FUNCTION_BLOCK FB_DO (* Service Interface Function Block Type *)
  (* Standard: 61499-2 *)
  (* Version 0.0, 2014-5-4, wildai, nxtControl GmbH, template *)
  (* Compiler Cpp nxtControl builtin 1.0 *)
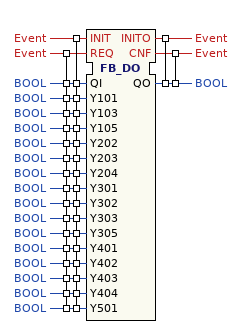
  EVENT_INPUT
    INIT WITH QI, Y101, Y103, Y105, Y202, Y203, Y204, Y301, Y302, Y303, Y305, Y401, Y402, Y403, Y404, Y501; (* Service Initialization *)
    REQ WITH QI, Y101, Y103, Y105, Y202, Y203, Y204, Y301, Y302, Y303, Y305, Y401, Y402, Y403, Y404, Y501; (* Service Request *)
  END_EVENT
  EVENT_OUTPUT
    INITO WITH QO; (* Initialization Confirm *)
    CNF WITH QO; (* Confirmation of Requested Service *)
  END_EVENT
  VAR_INPUT
    QI : BOOL; (* Event Input Qualifier *)
    Y101 : BOOL;
    Y103 : BOOL;
    Y105 : BOOL;
    Y202 : BOOL;
    Y203 : BOOL;
    Y204 : BOOL;
    Y301 : BOOL;
    Y302 : BOOL;
    Y303 : BOOL;
    Y305 : BOOL;
    Y401 : BOOL;
    Y402 : BOOL;
    Y403 : BOOL;
    Y404 : BOOL;
    Y501 : BOOL;
  END_VAR
  VAR_OUTPUT
    QO : BOOL; (* Event Output Qualifier *)
  END_VAR
  SERVICE FB_DO/RESOURCE
    SEQUENCE normal_establishment
      FB_DO.INIT+(PARAMS) -> RESOURCE.initialize(PARAMS) -> FB_DO.INITO+();
    END_SEQUENCE
    SEQUENCE unsuccessful_establishment
      FB_DO.INIT+(PARAMS) -> RESOURCE.initialize(PARAMS) -> FB_DO.INITO-(STATUS);
    END_SEQUENCE
    SEQUENCE request_confirm
      FB_DO.REQ+(SD) -> RESOURCE.request(SD) -> FB_DO.CNF+(RD);
    END_SEQUENCE
    SEQUENCE request_inhibited
      FB_DO.REQ-(SD) -> FB_DO.CNF-(STATUS);
    END_SEQUENCE
    SEQUENCE request_error
      FB_DO.REQ+(SD) -> RESOURCE.request(SD) -> FB_DO.CNF-(STATUS);
    END_SEQUENCE
    SEQUENCE indication_response
      FB_DO.RSP(QI,SD) -> RESOURCE.response(QI,SD);
      RESOURCE.indicate(RD) -> FB_DO.IND+(RD);
    END_SEQUENCE
    SEQUENCE indication_inhibited
      RESOURCE.indicate(RD,QI=FALSE) -> RESOURCE.inhibited();
    END_SEQUENCE
    SEQUENCE error_indication
      RESOURCE.error(STATUS) -> FB_DO.IND-(STATUS);
    END_SEQUENCE
    SEQUENCE application_initiated_termination
      FB_DO.INIT-() -> RESOURCE.terminate() -> FB_DO.INITO-(STATUS);
    END_SEQUENCE
    SEQUENCE resource_initiated_termination
      -> FB_DO.INITO-(STATUS);
    END_SEQUENCE
  END_SERVICE
END_FUNCTION_BLOCK
